// TIA Portal project "Task_4" (V18)

(* hardware
DEVICE "S7-1500/ET200MP station_1"  S7-1500 station
   slot 0: "导轨_0"  Rack  6ES7 590-1***0-0AA0
   slot 1: "PLC_1"  CPU 1516-3 PN/DP  6ES7 516-3AN01-0AB0  V2.6
      slot 3: "CPU 显示_1"  6ES7591-1BA00-0AA0
      slot 32768: "PROFINET 接口_1"  X1
      slot 33024: "PROFINET 接口_2"  X2
      slot 33280: "DP 接口_1"  X3
   slot 2: "DI 32x24VDC HF_1"  DI 32x24VDC HF  6ES7 521-1BL00-0AB0  V2.1
   slot 3: "DQ 32x24VDC/0.5A HF_1"  DQ 32x24VDC/0.5A HF  6ES7 522-1BL01-0AB0  V1.1
   slot 4: "AI 8xU/I/RTD/TC ST_1"  AI 8xU/I/RTD/TC ST  6ES7 531-7KF00-0AB0  V2.2
   slot 5: "AQ 4xU/I ST_1"  AQ 4xU/I ST  6ES7 532-5HD00-0AB0  V2.2
*)

// ===== PLC "PLC_1"  CPU 1516-3 PN/DP =====

VAR_GLOBAL   // PLC tag table "默认变量表"
   "按钮A次数" AT %MW100 : Int;
   "按钮A" AT %I1.0 : Bool;
   "按钮B" AT %I1.1 : Bool;
   "蓝灯" AT %Q1.0 : Bool;
   "Tag_1" AT %M10.0 : Bool;
END_VAR

// folder: System blocks/Program resources

DATA_BLOCK "T1"   // DB1
{ S7_Optimized_Access := 'TRUE' }
AUTHOR : Simatic
FAMILY : IEC
NAME : IEC_TMR
VERSION : 1.0
// stored: InstanceOfName IEC_TIMER
"IEC_TIMER"
BEGIN
END_DATA_BLOCK

// folder: (top level)

ORGANIZATION_BLOCK "Main"   // OB1, LAD, ProgramCycle
TITLE = "Main Program Sweep (Cycle)"
{ S7_Optimized_Access := 'TRUE' }
VERSION : 0.1
   VAR_INPUT
      Initial_Call : Bool;   // Initial call of this OB
      Remanence : Bool;   // =True, if remanent data are available
   END_VAR
   VAR_TEMP   // added for the SCL form of the ladder/FBD networks
      _w1 : Bool;
   END_VAR
BEGIN

REGION Network 1
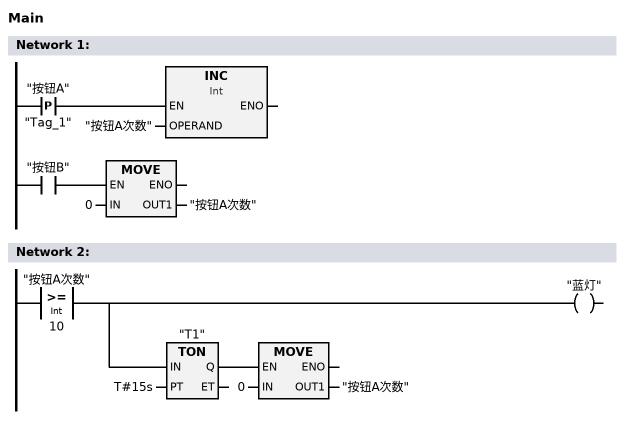
   RUNG wire#powerrail
      P_Contact(operand := "按钮A", bit := "Tag_1")
      { S7_Templates := "DestType := Int" } Inc( "按钮A次数" )
   END_RUNG
   RUNG wire#powerrail
      Contact( "按钮B" )
      Move(in := 0, out1 => "按钮A次数")
   END_RUNG
   // the same network as SCL:
   #_w1 := "按钮A" AND NOT "Tag_1";   // rising edge of "按钮A"
   "Tag_1" := "按钮A";
   IF #_w1 THEN "按钮A次数" := "按钮A次数" + 1; END_IF;
   IF "按钮B" THEN "按钮A次数" := 0; END_IF;
END_REGION

REGION Network 2
   "蓝灯" := "按钮A次数" >= 10;
   "T1".TON(IN := "蓝灯", PT := T#15s);
   IF "T1".Q THEN "按钮A次数" := 0; END_IF;
END_REGION
END_ORGANIZATION_BLOCK